ABB RobotStudio station: table with target.rsstn

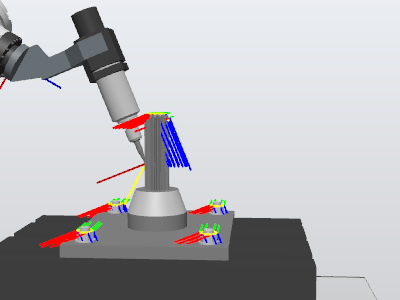
Station Station (saved by RobotStudio 22.3.10141.1)
Controller Controller11
  mechanical unit ROB_1: IRB1200_5_90_STD_03, 6 joints, base frame (0, 0, 0) mm
Layout (positions relative to the parent item):
  - IRB1200_5_90_STD_03 [mechanism, from %ABB.RobotStudio.Models.IRB1200%\IRB1200_5_90_STD_03.rslib] at (0, 0, 0) mm; joint values [0.2209, -0.1391, 0.8368, 4.0132, 0.2506, -3.8857] (rad or m)
  - MyTool [mechanism, from Training Objects\myTool.rslib] at (373.95, 68.03, 544.24) mm, rotated rx 180 ry 60 rz 180 deg
  - table_and_fixture_140 [part, from Training Objects\propeller_table.rslib] at (353.76, -152.36, 0) mm
Attachment: MyTool is attached to IRB1200_5_90_STD_03 / Link6
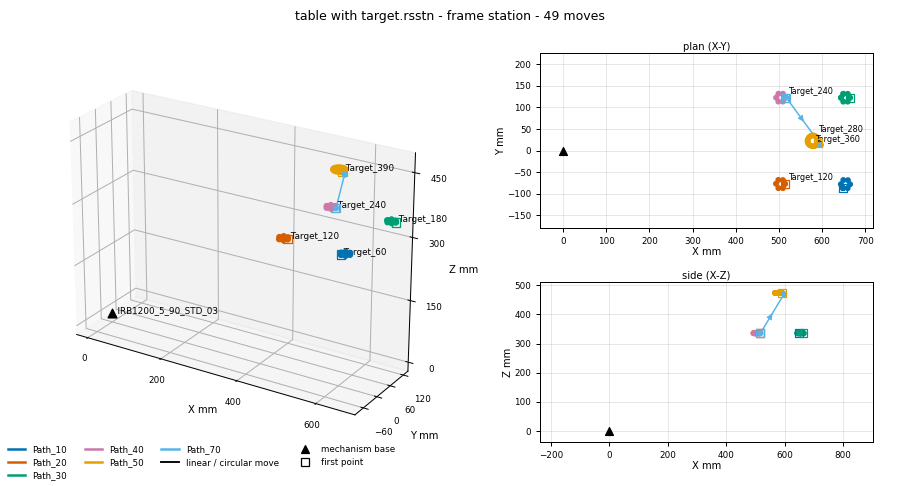
[picture p0: tool path of table with target.rsstn in frame station, 49 of 49 moves have a stored position in this frame; points joined in program order, loops and branches not executed]
Targets, tools, work objects and paths stored in the station, written as RAPID:
! task T_ROB1
MODULE CalibData
  PERS tooldata MyTool:=[TRUE,[[31.792631019,0,229.638935148],[0.945518576,0,0.325568154,0]],[1,[0,0,1],[1,0,0,0],0,0,0]];
ENDMODULE

! task T_ROB1
MODULE Module1
  CONST robtarget Target_10:=[[643.274341562,-77.587869859,335.337177029],[0.190808171,0.000000673,0.981627344,0.000000554],[-1,1,-2,0],[9E+09,9E+09,9E+09,9E+09,9E+09,9E+09]];
  CONST robtarget Target_20:=[[648.89660735,-68.057368816,335.337082934],[0.190807942,0.000000682,0.981627388,0.00000059],[-1,1,-2,0],[9E+09,9E+09,9E+09,9E+09,9E+09,9E+09]];
  CONST robtarget Target_30:=[[659.546396875,-68.404653242,335.337072517],[0.190807525,0.00000062,0.981627469,0.00000057],[-1,1,-2,0],[9E+09,9E+09,9E+09,9E+09,9E+09,9E+09]];
  CONST robtarget Target_40:=[[664.448404148,-77.73676707,335.337077819],[0.190807241,0.000000583,0.981627524,0.000000544],[-1,1,-2,0],[9E+09,9E+09,9E+09,9E+09,9E+09,9E+09]];
  CONST robtarget Target_50:=[[659.00251017,-86.693660366,335.337076188],[0.190806945,0.000000654,0.981627582,0.00000061],[-1,1,-2,0],[9E+09,9E+09,9E+09,9E+09,9E+09,9E+09]];
  CONST robtarget Target_60:=[[648.378819952,-86.693651882,335.337082741],[0.19080676,0.000000604,0.981627618,0.000000583],[-1,1,-2,0],[9E+09,9E+09,9E+09,9E+09,9E+09,9E+09]];
  CONST robtarget Target_70:=[[509.145034318,-86.693616566,335.336971563],[0.190806541,0.000000577,0.981627661,0.000000598],[-1,1,-2,0],[9E+09,9E+09,9E+09,9E+09,9E+09,9E+09]];
  CONST robtarget Target_80:=[[498.59071844,-86.693606879,335.336968434],[0.190806449,0.000000638,0.981627678,0.000000648],[-1,1,-2,0],[9E+09,9E+09,9E+09,9E+09,9E+09,9E+09]];
  CONST robtarget Target_90:=[[493.061918752,-76.502313306,335.336976884],[0.190805831,0.000000682,0.981627799,0.000000718],[-1,1,-2,0],[9E+09,9E+09,9E+09,9E+09,9E+09,9E+09]];
  CONST robtarget Target_100:=[[498.533905874,-67.753039265,335.336952313],[0.190805219,0.000000618,0.981627917,0.000000748],[-1,1,-2,0],[9E+09,9E+09,9E+09,9E+09,9E+09,9E+09]];
  CONST robtarget Target_110:=[[509.10439372,-68.160486042,335.336981028],[0.190804837,0.000000634,0.981627992,0.000000784],[-1,1,-2,0],[9E+09,9E+09,9E+09,9E+09,9E+09,9E+09]];
  CONST robtarget Target_120:=[[513.793185591,-76.926688182,335.199346378],[0.190804234,0.000000469,0.981628109,0.00000069],[-1,1,-2,0],[9E+09,9E+09,9E+09,9E+09,9E+09,9E+09]];
  CONST robtarget Target_130:=[[659.016094731,113.502704134,335.199262556],[0.190803839,0.000000628,0.981628186,0.000000831],[0,2,-3,0],[9E+09,9E+09,9E+09,9E+09,9E+09,9E+09]];
  CONST robtarget Target_140:=[[648.773106814,113.478385383,335.199069853],[0.190802054,0.000000959,0.981628533,0.00000105],[0,2,-3,0],[9E+09,9E+09,9E+09,9E+09,9E+09,9E+09]];
  CONST robtarget Target_150:=[[643.512143752,122.544591829,335.199045692],[0.190801825,0.000000976,0.981628577,0.000001074],[0,2,-3,0],[9E+09,9E+09,9E+09,9E+09,9E+09,9E+09]];
  CONST robtarget Target_160:=[[648.820835483,131.48089695,334.930564814],[0.190800554,0.000001058,0.981628824,0.000001117],[0,2,-3,0],[9E+09,9E+09,9E+09,9E+09,9E+09,9E+09]];
  CONST robtarget Target_170:=[[659.182815687,131.4809055,334.930578126],[0.190800458,0.000001139,0.981628843,0.000001189],[0,2,-3,0],[9E+09,9E+09,9E+09,9E+09,9E+09,9E+09]];
  CONST robtarget Target_180:=[[664.197692397,122.523782928,335.196064354],[0.190799432,0.000001291,0.981629042,0.00000129],[0,2,-3,0],[9E+09,9E+09,9E+09,9E+09,9E+09,9E+09]];
  CONST robtarget Target_190:=[[508.962531806,131.691782122,335.07525232],[0.190797523,0.000001928,0.981629413,0.000001823],[0,2,-3,0],[9E+09,9E+09,9E+09,9E+09,9E+09,9E+09]];
  CONST robtarget Target_200:=[[498.608227395,131.691817076,335.075264802],[0.190797383,0.000001796,0.981629441,0.000001775],[0,2,-3,0],[9E+09,9E+09,9E+09,9E+09,9E+09,9E+09]];
  CONST robtarget Target_210:=[[493.362209574,122.688909811,335.075163631],[0.190797134,0.00000172,0.981629489,0.000001749],[0,2,-3,0],[9E+09,9E+09,9E+09,9E+09,9E+09,9E+09]];
  CONST robtarget Target_220:=[[498.544627244,113.644188186,335.075167429],[0.190797039,0.000001665,0.981629507,0.000001759],[0,2,-3,0],[9E+09,9E+09,9E+09,9E+09,9E+09,9E+09]];
  CONST robtarget Target_230:=[[508.975343557,113.644209344,335.075160978],[0.190796738,0.000001647,0.981629566,0.00000174],[0,2,-3,0],[9E+09,9E+09,9E+09,9E+09,9E+09,9E+09]];
  CONST robtarget Target_240:=[[513.951148517,122.745672769,335.0750771],[0.190796422,0.000001784,0.981629627,0.000001767],[0,2,-3,0],[9E+09,9E+09,9E+09,9E+09,9E+09,9E+09]];
  CONST robtarget Target_250:=[[591.19303994,21.3303063,472.999954045],[0.19079594,0.000001778,0.981629721,0.000001752],[0,1,-2,1],[9E+09,9E+09,9E+09,9E+09,9E+09,9E+09]];
  CONST robtarget Target_260:=[[590.649750447,26.499632421,472.999963889],[0.190795845,0.000001772,0.98162974,0.000001748],[0,1,-2,1],[9E+09,9E+09,9E+09,9E+09,9E+09,9E+09]];
  CONST robtarget Target_270:=[[587.627611886,31.448387931,472.999950087],[0.190795734,0.000001762,0.981629761,0.000001736],[0,1,-2,1],[9E+09,9E+09,9E+09,9E+09,9E+09,9E+09]];
  CONST robtarget Target_280:=[[583.277128488,34.292766814,472.999953903],[0.190795641,0.000001743,0.981629779,0.000001712],[0,1,-2,1],[9E+09,9E+09,9E+09,9E+09,9E+09,9E+09]];
  CONST robtarget Target_290:=[[579.357060623,35.126018203,472.999972738],[0.190795552,0.000001741,0.981629796,0.00000171],[0,1,-2,1],[9E+09,9E+09,9E+09,9E+09,9E+09,9E+09]];
  CONST robtarget Target_300:=[[573.677207245,34.056244117,472.999955552],[0.19079554,0.000001735,0.981629799,0.000001705],[0,1,-2,1],[9E+09,9E+09,9E+09,9E+09,9E+09,9E+09]];
  CONST robtarget Target_310:=[[569.472108392,31.001051353,472.999971802],[0.190795452,0.000001739,0.981629816,0.000001711],[0,1,-2,1],[9E+09,9E+09,9E+09,9E+09,9E+09,9E+09]];
  CONST robtarget Target_320:=[[566.873342165,26.499629319,472.999969149],[0.19079545,0.000001743,0.981629816,0.000001712],[0,1,-2,1],[9E+09,9E+09,9E+09,9E+09,9E+09,9E+09]];
  CONST robtarget Target_330:=[[566.125531011,21.998358206,472.999944842],[0.190795433,0.000001729,0.98162982,0.000001695],[0,1,-2,1],[9E+09,9E+09,9E+09,9E+09,9E+09,9E+09]];
  CONST robtarget Target_340:=[[567.477617971,16.9140493,472.999973919],[0.190795366,0.000001719,0.981629833,0.000001685],[0,1,-2,1],[9E+09,9E+09,9E+09,9E+09,9E+09,9E+09]];
  CONST robtarget Target_350:=[[570.925027695,12.898321215,472.999966116],[0.190795361,0.000001729,0.981629834,0.000001696],[0,1,-2,1],[9E+09,9E+09,9E+09,9E+09,9E+09,9E+09]];
  CONST robtarget Target_360:=[[576.162594564,10.410069603,472.999946934],[0.190795347,0.000001725,0.981629836,0.000001693],[0,1,-2,1],[9E+09,9E+09,9E+09,9E+09,9E+09,9E+09]];
  CONST robtarget Target_370:=[[581.360312117,10.410068925,472.999974358],[0.190795268,0.000001712,0.981629852,0.000001677],[0,1,-2,1],[9E+09,9E+09,9E+09,9E+09,9E+09,9E+09]];
  CONST robtarget Target_380:=[[586.742010363,12.819277393,472.999960672],[0.190795258,0.000001688,0.981629854,0.00000165],[0,1,-2,1],[9E+09,9E+09,9E+09,9E+09,9E+09,9E+09]];
  CONST robtarget Target_390:=[[590.045289361,16.914049315,472.999944524],[0.190795246,0.000001698,0.981629856,0.000001662],[0,1,-2,1],[9E+09,9E+09,9E+09,9E+09,9E+09,9E+09]];
  CONST robtarget Target_400:=[[516.784350791,122.745723171,335.075099713],[0.190796151,0.000001769,0.98162968,0.000001807],[0,2,-3,0],[9E+09,9E+09,9E+09,9E+09,9E+09,9E+09]];
  CONST robtarget Target_410:=[[597.061293702,13.320911106,468.689370264],[0.190795249,0.000002096,0.981629855,0.00000223],[0,2,-3,0],[9E+09,9E+09,9E+09,9E+09,9E+09,9E+09]];
  PROC Path_10()
    MoveL Target_60,v1000,fine,MyTool\WObj:=wobj0;
    MoveL Target_10,v1000,fine,MyTool\WObj:=wobj0;
    MoveL Target_20,v1000,fine,MyTool\WObj:=wobj0;
    MoveL Target_30,v1000,fine,MyTool\WObj:=wobj0;
    MoveL Target_40,v1000,fine,MyTool\WObj:=wobj0;
    MoveL Target_50,v1000,fine,MyTool\WObj:=wobj0;
    MoveL Target_60,v1000,fine,MyTool\WObj:=wobj0;
    MoveL Target_60,v1000,fine,MyTool\WObj:=wobj0;
  ENDPROC
  PROC Path_20()
    MoveL Target_120,v1000,fine,MyTool\WObj:=wobj0;
    MoveL Target_70,v1000,fine,MyTool\WObj:=wobj0;
    MoveL Target_80,v1000,fine,MyTool\WObj:=wobj0;
    MoveL Target_90,v1000,fine,MyTool\WObj:=wobj0;
    MoveL Target_100,v1000,fine,MyTool\WObj:=wobj0;
    MoveL Target_110,v1000,fine,MyTool\WObj:=wobj0;
    MoveL Target_120,v1000,fine,MyTool\WObj:=wobj0;
  ENDPROC
  PROC Path_30()
    MoveL Target_180,v1000,fine,MyTool\WObj:=wobj0;
    MoveL Target_130,v1000,fine,MyTool\WObj:=wobj0;
    MoveL Target_140,v1000,fine,MyTool\WObj:=wobj0;
    MoveL Target_150,v1000,fine,MyTool\WObj:=wobj0;
    MoveL Target_150,v1000,fine,MyTool\WObj:=wobj0;
    MoveL Target_160,v1000,fine,MyTool\WObj:=wobj0;
    MoveL Target_160,v1000,fine,MyTool\WObj:=wobj0;
    MoveL Target_170,v1000,fine,MyTool\WObj:=wobj0;
    MoveL Target_180,v1000,fine,MyTool\WObj:=wobj0;
  ENDPROC
  PROC Path_40()
    MoveL Target_240,v1000,fine,MyTool\WObj:=wobj0;
    MoveL Target_190,v1000,fine,MyTool\WObj:=wobj0;
    MoveL Target_200,v1000,fine,MyTool\WObj:=wobj0;
    MoveL Target_210,v1000,fine,MyTool\WObj:=wobj0;
    MoveL Target_220,v1000,fine,MyTool\WObj:=wobj0;
    MoveL Target_230,v1000,fine,MyTool\WObj:=wobj0;
    MoveL Target_240,v1000,fine,MyTool\WObj:=wobj0;
  ENDPROC
  PROC Path_50()
    MoveL Target_390,v1000,z100,MyTool\WObj:=wobj0;
    MoveL Target_250,v1000,z100,MyTool\WObj:=wobj0;
    MoveL Target_260,v1000,z100,MyTool\WObj:=wobj0;
    MoveL Target_270,v1000,z100,MyTool\WObj:=wobj0;
    MoveL Target_280,v1000,z100,MyTool\WObj:=wobj0;
    MoveL Target_290,v1000,z100,MyTool\WObj:=wobj0;
    MoveL Target_300,v1000,z100,MyTool\WObj:=wobj0;
    MoveL Target_310,v1000,z100,MyTool\WObj:=wobj0;
    MoveL Target_320,v1000,z100,MyTool\WObj:=wobj0;
    MoveL Target_330,v1000,z100,MyTool\WObj:=wobj0;
    MoveL Target_340,v1000,z100,MyTool\WObj:=wobj0;
    MoveL Target_350,v1000,z100,MyTool\WObj:=wobj0;
    MoveL Target_360,v1000,z100,MyTool\WObj:=wobj0;
    MoveL Target_370,v1000,z100,MyTool\WObj:=wobj0;
    MoveL Target_380,v1000,z100,MyTool\WObj:=wobj0;
    MoveL Target_390,v1000,z100,MyTool\WObj:=wobj0;
    Path_70;
    Path_70;
    Path_70;
    Path_70;
    Path_70;
  ENDPROC
  PROC Path_60()
    Path_10;
    Path_20;
    Path_30;
    Path_40;
    Path_70;
    Path_50;
  ENDPROC
  PROC Path_70()
    MoveL Target_400,v1000,z100,MyTool\WObj:=wobj0;
    MoveL Target_410,v1000,z100,MyTool\WObj:=wobj0;
  ENDPROC
ENDMODULE

